SUBAPPLICATION AX_SUBSCRIBE_BG_OPC (* OPC-UA Remote-Subscribe + VT-Hintergrundfarbe (generisch, ein Kanal) *)
  (* Standard: 61499-2 *)
  (* Version 1.1, 2026-09-27, Franz Höpfinger, Meisterschulen am Ostbahnhof, Neuer Plug OUT (lokal) - bisher verliess der abonnierte Wert diesen Typ nur in die eigene Hintergrundfarbe, kein lokaler Zugriff fuer weitere Konsumenten moeglich (z.B. Bunkerboden-Gruen-Feedback braucht 'Bunker ausgeklappt' zusaetzlich zur eigenen IO-Grid-Anzeige). AX_SUBSCRIBE_1.OUT jetzt per neuem AX_SPLIT_2 auf GreenWhiteBackground1_AX UND OUT verzweigt. *)
  (* Version 1.0, 2026-08-27, franz, Meisterschulen am Ostbahnhof *)
  PACKAGE MyLib::sys;
  IMPORT isobus::UT::Q::const::IDs::ID_NULL;
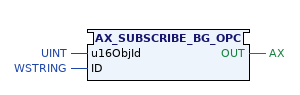
  VAR_INPUT
    u16ObjId : UINT := ID_NULL; (* Object ID Hintergrund-Rechteck (VT) *)
    ID : WSTRING; (* OPC-UA Remote-Subscribe-Adresse *)
  END_VAR
  PLUGS
    OUT : adapter::types::unidirectional::AX; (* Abonnierter Wert, lokal - fuer Weiterverarbeitung ohne zweiten Self-Subscribe desselben Knotens *)
  END_PLUGS
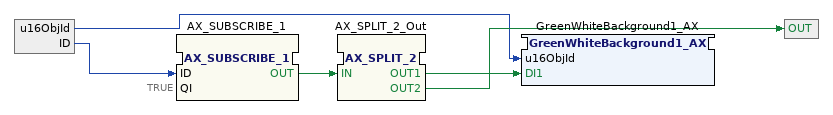
  FBS
    AX_SUBSCRIBE_1 : adapter::net::AX_SUBSCRIBE_1(QI := TRUE);
    AX_SPLIT_2_Out : adapter::events::unidirectional::AX_SPLIT_2;
  END_FBS
  SUBAPPS
    GreenWhiteBackground1_AX : MyLib::sys::GreenWhiteBackground1_AX;
  END_SUBAPPS
  DATA_CONNECTIONS
    ID TO AX_SUBSCRIBE_1.ID;
    u16ObjId TO GreenWhiteBackground1_AX.u16ObjId;
  END_CONNECTIONS
  ADAPTER_CONNECTIONS
    AX_SUBSCRIBE_1.OUT TO AX_SPLIT_2_Out.IN;
    AX_SPLIT_2_Out.OUT1 TO GreenWhiteBackground1_AX.DI1;
    AX_SPLIT_2_Out.OUT2 TO OUT;
  END_CONNECTIONS
END_SUBAPPLICATION
